// TwinCAT 3 PLC project HelloWorld
// ProgramVersion: 3.1.4024.0
// libraries:
//   Tc2_Standard, * (Beckhoff Automation GmbH)
//   Tc2_System, * (Beckhoff Automation GmbH)
//   Tc2_Utilities, * (Beckhoff Automation GmbH)
//   Tc3_Module, * (Beckhoff Automation GmbH)
// project tree:
//   DUTs/ E_Color.TcDUT, E_Event.TcDUT, ST_Event.TcDUT, ST_Student.TcDUT
//   GVLs/ Nums.TcGVL
//   / PlcTask.TcTTO
//   POUs/ Celcius_Fahrenheit.TcPOU, F_Add.TcPOU, F_InitializeStudentDetails.TcPOU, F_Loops.TcPOU, F_Multiply.TcPOU, F_PrimeCheck.TcPOU, F_UpdateTimeWithSystemTime.TcPOU, F_HelloWorld.TcPOU, MAIN.TcPOU
// real-time tasks:
//   TASK PlcTask: cycle T#10ms, priority 20, ADS port 350
//   TASK PlcTask1: cycle T#10ms, priority 21, ADS port 351

CONFIGURATION HelloWorld
    RESOURCE PLC ON TwinCAT3
        TASK PlcTask(INTERVAL := T#10ms, PRIORITY := 20);
        PROGRAM MAIN WITH PlcTask : MAIN;
    END_RESOURCE
END_CONFIGURATION

// ---- DUTs/E_Color.TcDUT
{attribute 'qualified_only'}
{attribute 'strict'}
TYPE E_Color :
(
	Red := 0,
	Blue := 1,
	Green:= 2
);
END_TYPE

// ---- DUTs/E_Event.TcDUT
{attribute 'qualified_only'}
{attribute 'strict'}
TYPE E_Event :
(
	Alarm := 0,
	Message := 1
);
END_TYPE

// ---- DUTs/ST_Event.TcDUT
TYPE ST_Event :
STRUCT
	eEventType : E_Event;
	eEventSeverity : TcEventSeverity;
	nEventIdentity : UDINT;
	sEventText : STRING(255);
	dtTimestamp : DATE_AND_TIME;
END_STRUCT
END_TYPE

// ---- DUTs/ST_Student.TcDUT
TYPE ST_Student :
STRUCT
	sStudentName : STRING(255);
	nStudentId : INT;
	nStudentAge : INT;
END_STRUCT
END_TYPE

// ---- GVLs/Nums.TcGVL
{attribute 'qualified_only'}
VAR_GLOBAL
END_VAR

// ---- POUs/MAIN.TcPOU
PROGRAM MAIN
VAR
	fFahrenheit : REAL;
	stEventOne : ST_Event;
	bFlag : BOOL := FALSE;
	nSum : INT;
	nProd : DINT;
	bIsPrime : BOOL;
	nResultFromLoop1 : INT;
	nResultFromLoop2 : INT;
	nResultFromLoop3 : INT;
	
	stStudentReference1 : ST_Student;
END_VAR


IF NOT bFlag THEN 
fFahrenheit := Celcius_Fahrenheit(fCelcius := 5.0);
F_UpdateTimeWithSystemTime(stEventOne);
F_Add(nFirstNum:= 29, nSecondNum:= 32,nResult => nSum );
bFlag := TRUE;
nProd := F_Multiply(123,432);
bIsPrime := F_PrimeCheck(nInputNum := 17 );

F_InitializeStudentDetails(stStudentReference1, 'Kamesh', 101 , 21);

F_Loops(10,nResult1 => nResultFromLoop1, nResult2 => nResultFromLoop2, nResult3 => nResultFromLoop3);

END_IF

END_PROGRAM

// ---- POUs/Celcius_Fahrenheit.TcPOU
FUNCTION Celcius_Fahrenheit : REAL
VAR_INPUT
	fCelcius : REAL;
END_VAR
VAR
END_VAR

Celcius_Fahrenheit := fCelcius * 1.8 + 32.0;

END_FUNCTION

// ---- POUs/F_UpdateTimeWithSystemTime.TcPOU
FUNCTION F_UpdateTimeWithSystemTime
VAR_INPUT
	stEvent : REFERENCE TO ST_Event;
END_VAR
VAR
	fbGETSYSTEMTIME : GETSYSTEMTIME;
	stFileTime : T_FILETIME;
END_VAR

fbGETSYSTEMTIME(timeLoDW => stFileTime.dwLowDateTime,
				timeHiDW => stFileTime.dwHighDateTime);
stEvent.dtTimestamp := FILETIME_TO_DT(fileTime := stFileTime);

END_FUNCTION

// ---- POUs/F_Add.TcPOU
FUNCTION F_Add : INT
VAR_INPUT
	nFirstNum : INT;
	nSecondNum : INT;
END_VAR
VAR_OUTPUT
	nResult : INT;
END_VAR
VAR
END_VAR

nResult := nFirstNum + nSecondNum;

END_FUNCTION

// ---- POUs/F_Multiply.TcPOU
FUNCTION F_Multiply : DINT
VAR_INPUT
	nNum1 : INT;
	nNum2 : INT;
END_VAR
VAR
END_VAR

F_Multiply := nNum1 * nNum2;

END_FUNCTION

// ---- POUs/F_PrimeCheck.TcPOU
FUNCTION F_PrimeCheck : BOOL
VAR_INPUT
	nInputNum : INT;
	
END_VAR

VAR
	nLimit : INT;
	nIterator : INT;
END_VAR


F_PrimeCheck := TRUE;
IF nInputNum > 1 THEN
	nLimit := nInputNum/2;
	FOR nIterator := 2 TO nLimit  DO
		IF (nInputNum MOD nIterator) = 0 THEN 
			F_PrimeCheck := FALSE;
			EXIT;
		END_IF
	END_FOR
END_IF
IF nInputNum <=1 THEN 
	F_PrimeCheck := FALSE;
	RETURN;
END_IF

END_FUNCTION

// ---- POUs/F_InitializeStudentDetails.TcPOU
FUNCTION F_InitializeStudentDetails
VAR_INPUT
	stStudent1 : REFERENCE TO ST_Student;
	stName : STRING(255);
	stId : INT;
	stAge :INT;
END_VAR
VAR
END_VAR

stStudent1.sStudentName := stName;
stStudent1.nStudentAge := stAge;
stStudent1.nStudentId := stId;

END_FUNCTION

// ---- POUs/F_Loops.TcPOU
FUNCTION F_Loops : INT 
VAR_INPUT
	nInputNum1 : INT;
END_VAR
VAR_OUTPUT
	nResult1 : INT;
	nResult2 : INT;
	nResult3 : INT;
END_VAR
VAR
	nCounter : INT;
END_VAR

FOR nCounter := 1 TO nInputNum1 DO
	nResult1 := nResult1 + nCounter;
END_FOR

nInputNum1 := 1;
WHILE nInputNum1 <> 10 DO
	nInputNum1 := nInputNum1 + 1;
	nResult2 := nResult2 + nInputNum1;
END_WHILE

nCounter := 0;
REPEAT
	nCounter := nCounter + 1;
	nResult3 := nResult3 + nCounter;
	
	UNTIL
	nCounter = 10
END_REPEAT

END_FUNCTION

// ---- POUs/F_HelloWorld.TcPOU
FUNCTION F_HelloWorld
VAR_INPUT
END_VAR
VAR
	run: BOOL;
END_VAR

IF NOT run THEN
		ADSLOGSTR(msgCtrlMask := ADSLOG_MSGTYPE_ERROR OR ADSLOG_MSGTYPE_LOG,
			msgFmtStr:= 'Hello world!!',
			strArg:='');
			
		run := TRUE;
END_IF

END_FUNCTION
